(* PLC project Unnamed, Unknown Unnamed 1 *)
(* stored: creationDateTime 2025-11-07T11:54:43, modificationDateTime 2025-11-14T14:02:27 *)

TYPE datatype0 : BOOL;
END_TYPE

PROGRAM latch
  VAR
    start : BOOL := True;
    stop : BOOL;
    moteur : BOOL;
  END_VAR

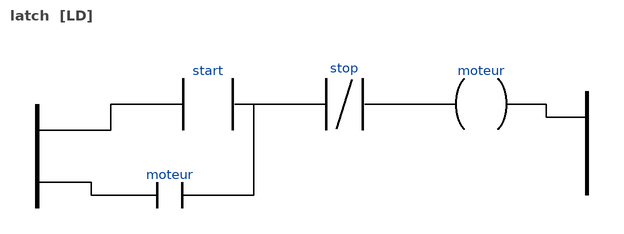
(* LD diagram, written out as Structured Text *)
moteur := (start OR moteur) AND NOT stop;
END_PROGRAM

PROGRAM setreset
  VAR
    SET : BOOL;
    RESET : BOOL;
    MOTOR : BOOL;
    RS0 : RS;
  END_VAR

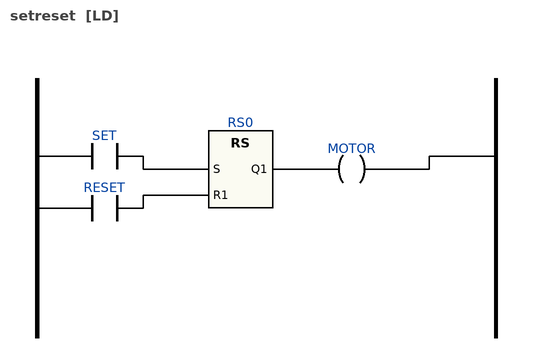
(* LD diagram, written out as Structured Text *)
RS0(S := SET, R1 := RESET);
MOTOR := RS0.Q1;
END_PROGRAM

PROGRAM temp
  VAR
    SET : BOOL;
    RESET : BOOL;
    TON1 : TIME := T#100ms;
    RS0 : RS;
    TON0 : TON;
  END_VAR

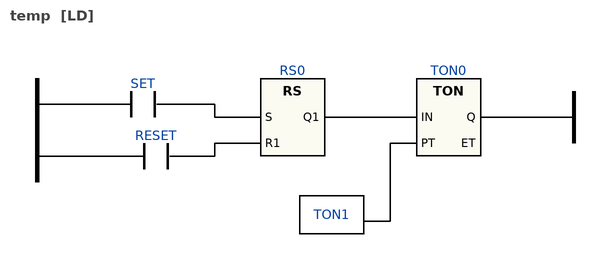
(* LD diagram, written out as Structured Text *)
RS0(S := SET, R1 := RESET);
TON0(IN := RS0.Q1, PT := TON1);
END_PROGRAM

CONFIGURATION Config0
  RESOURCE Res0 ON PLC
    TASK task0(INTERVAL := T#20ms, PRIORITY := 0);
    PROGRAM instance0 WITH task0 : setreset;
  END_RESOURCE
END_CONFIGURATION
